FUNCTION_BLOCK FB_Debounce
VAR_INPUT
	tOnDelay	: TIME;
	tOffDelay	: TIME;
	xRawSignal	: BOOL;
END_VAR
VAR_OUTPUT
	Debounced	: BOOL;
END_VAR
VAR
	TimerOn 	: Tc2_Standard.TON;
	TimerOff 	: Tc2_Standard.TOF;
	ftSignal	: Tc2_Standard.F_TRIG;
END_VAR

TimerOn(PT := tOnDelay);  //TON
TimerOff(PT := tOffDelay);  //TOF
ftSignal(CLK := xRawSignal);

TimerOn.IN := xRawSignal;
TimerOff.IN := ftSignal.Q; 

Debounced := TimerOn.Q OR TimerOff.Q;

END_FUNCTION_BLOCK

(* stored: Version 1.1.0.1
   POU FB_Debounce: Id {5c414ebf-65a9-0af7-23b2-89a791f4af19}, SpecialFunc None *)
